(* CoDeSys 2.3.9.35 project: semaforo.pro *)
(* Author: Altus *)
(* Libraries: DU35x.lib 7.7.11 15:59:13, Navigation.lib 15.7.11 10:06:00, SysLibTargetVisu.lib 26.11.08 09:53:28, Standard.lib 26.11.08 09:46:20, Iecsfc.lib 26.11.08 09:46:14, SYSLIBCALLBACK.LIB 26.11.08 09:53:30 *)

(* PLC configuration (modules and I/O channels)
COM1 [COM1] node 0, in %IB0 out %QB0 {BaudRate = 115200; Paridade = Sem Paridade; StopBits = 1 Stop Bit; Modem = Sem RTS/CTS; Delay = 5}
  MODBUS Escravo [Escravo] node 0, in %IB0 out %QB0 {EnderecoModbus = 2}
COM2 [COM2] node 1, in %IB0 out %QB0 {BaudRate = 115200; Paridade = Sem Paridade; StopBits = 1 Stop Bit; Modem = Sem RTS/CTS; Delay = 5}
  Desabilitada [Desabilitado485] node 0, in %IB0 out %QB0
Barramento [Barramento] node 1, in %IB0 out %QB0
  Entradas [Entradas] node 0, in %IB0 out %QB0
    Entradas Digitais 0 [Entradas0] node 0, in %IW0 out %QB0
      I00 AT %IX0.0 [BitInput] I0.0
      I01 AT %IX0.1 [BitInput] I0.1
      I02 AT %IX0.2 [BitInput] I0.2
      I03 AT %IX0.3 [BitInput] I0.3
      I04 AT %IX0.4 [BitInput] I0.4
      I05 AT %IX0.5 [BitInput] I0.5
      I06 AT %IX0.6 [BitInput] I0.6
      I07 AT %IX0.7 [BitInput] I0.7
      I08 AT %IX0.8 [BitInput] I0.8
    Entradas Digitais 1 [Entradas1] node 0, in %IW1 out %QB0
      I10 AT %IX1.0 [BitInput] I1.0
      I11 AT %IX1.1 [BitInput] I1.1
      I12 AT %IX1.2 [BitInput] I1.2
      I13 AT %IX1.3 [BitInput] I1.3
      I14 AT %IX1.4 [BitInput] I1.4
      I15 AT %IX1.5 [BitInput] I1.5
      I16 AT %IX1.6 [BitInput] I1.6
      I17 AT %IX1.7 [BitInput] I1.7
      I18 AT %IX1.8 [BitInput] I1.8
    Entradas Digitais 2 [Entradas2] node 0, in %IW2 out %QB0
      I20 AT %IX2.0 [BitInput] I2.0
      I21 AT %IX2.1 [BitInput] I2.1
    Entradas Analógicas [EntradaAnalogica] node 0, in %IW4 out %QB0
      AI0 AT %IW4 [WordInput] AI0 {TipoAnalogica = Channel Disable; FiltroAnalogica = Filter 0 - AI=2ms  / AV=90ms; FundoEscala = 0}
      AI1 AT %IW5 [WordInput] AI1 {TipoAnalogica = Channel Disable; FiltroAnalogica = Filter 0 - AI=2ms  / AV=90ms; FundoEscala = 0}
      AI2 AT %IW6 [WordInput] AI2 {TipoAnalogica = Channel Disable; FiltroAnalogica = Filter 0 - AI=2ms  / AV=90ms; FundoEscala = 0}
      AI3 AT %IW7 [WordInput] AI3 {TipoAnalogica = Channel Disable; FiltroAnalogica = Filter 0 - AI=2ms  / AV=90ms; FundoEscala = 0}
    Entradas Rápidas [EntradasRapidas] node 1, in %IB16 out %QB0
      Bloco 0 [Bloco0] node 0, in %IB16 out %QB0
        Desabilitado [DesabilitadoBloco0] node 0, in %IB16 out %QB0
      Bloco 1 [Bloco1] node 1, in %IB16 out %QB0
        Desabilitado [DesabilitadoBloco1] node 0, in %IB16 out %QB0
      Entrada Configuravél Bloco 0 [EntradaConfiBloco0] node 2, in %IB16 out %QB0
        Contador 0 [EntradaConfContador0] node 0, in %IB16 out %QB0 {EntradaConfiguravelContador = Disable}
      Entrada Configuravél Bloco 1 [EntradaConfiBloco1] node 3, in %IB16 out %QB0
        Contador 2 [EntradaConfContador2] node 0, in %IB16 out %QB0 {EntradaConfiguravelContador = Disable}
  Saídas [Saidas] node 1, in %IB13 out %QB0
    Saídas Digitais 0 [Saidas0] node 0, in %IW0 out %QW0
      Q00 AT %QX0.0 [BitOutput] Q0.0
      Q01 AT %QX0.1 [BitOutput] Q0.1
      Q02 AT %QX0.2 [BitOutput] Q0.2
      Q03 AT %QX0.3 [BitOutput] Q0.3
      Q04 AT %QX0.4 [BitOutput] Q0.4
      Q05 AT %QX0.5 [BitOutput] Q0.5
      Q06 AT %QX0.6 [BitOutput] Q0.6
      Q07 AT %QX0.7 [BitOutput] Q0.7
    Saídas Digitais 1 [Saidas1] node 0, in %IW0 out %QW1
      Q10 AT %QX1.0 [BitOutput] Q1.0
      Q11 AT %QX1.1 [BitOutput] Q1.1
      Q12 AT %QX1.2 [BitOutput] Q1.2
      Q13 AT %QX1.3 [BitOutput] Q1.3
      Q14 AT %QX1.4 [BitOutput] Q1.4
      Q15 AT %QX1.5 [BitOutput] Q1.5
      Q16 AT %QX1.6 [BitOutput] Q1.6
      Q17 AT %QX1.7 [BitOutput] Q1.7
    Saídas Analógicas [SaidaAnalogica] node 0, in %IW0 out %QW3
      AO0 AT %QW3 [WordOutput] AO0 {TipoAnalogica = Channel Disable; FundoEscala = 0}
      AO1 AT %QW4 [WordOutput] AO1 {TipoAnalogica = Channel Disable; FundoEscala = 0}
    Saídas Rápidas [SaidasRapidas] node 1, in %IB0 out %QB10
      Saída Rápida 0 Desabilitada [DesabilitadoF0] node 0, in %IB0 out %QB10
      Saída Rápida 1 Desabilitada [DesabilitadoF1] node 1, in %IB0 out %QB10
    Saídas Comum de Contador [SaidasContador] node 2, in %IB0 out %QB10
      Saída do Bloco 0 Desabilitada [DesabilitadoSaidaBloco0] node 0, in %IB0 out %QB10
      Saída do Bloco 1 Desabilitada [DesabilitadoSaidaBloco1] node 1, in %IB0 out %QB10
Eventos Externos [Eventos] node 2, in %IB13 out %QB6
  Evento Temporizado [TimerEvent] node 0, in %IB13 out %QB6 {Intervalo = 10}
*)

(* Task configuration *)
TASK PRINCIPAL (PRIORITY := 1, INTERVAL := T#100ms);
	PLC_PRG();
END_TASK
TASK NAVIGATION (PRIORITY := 1, INTERVAL := T#20ms);
	NAVEGA();
END_TASK
TASK VISUALIZATION (PRIORITY := 1, INTERVAL := T#500ms);
	MAINTARGETVISU_PAINT_CODE
END_TASK
TASK KEYBOARD_USAGE (PRIORITY := 1, INTERVAL := T#20ms);
	MAINTARGETVISU_INPUT_CODE
END_TASK

(* POU PLC_PRG, LD *)
PROGRAM PLC_PRG
VAR
	t1: TON;
	t2: TON;
	t3: TON;
	t4: TON;
	t5: TON;
	t6: TON;
	v1: TON;
	a1: TON;
	ton1: TON;
	aux1: BOOL;
	taux: TON;
	vermelho_in AT %MW3: WORD;
	verde_in AT %MW4: WORD;
	amarelo_in : REAL := 4000;
	vermelho_out: TIME;
	verde_out: TIME;
	amarelo_out: TIME;
	RED: DWORD;
	Defeito: BOOL;
	td: TON;
	S_def: BOOL;
	td2: TON;
	S_def2: BOOL;
	t7: TON;
	t8: TON;
	t9: TON;
	t10: TON;
	t11: TON;
	t12: TON;
	td3: TON;
	td4: TON;
	auxv2: BOOL;
	a2: TON;
	auxa2: BOOL;
	aux_t7: BOOL;
	aux_t8: BOOL;
	aux_t9: BOOL;
	aux_t10: BOOL;
	t_aux11: BOOL;
	aux_t12: BOOL;
	bob: BOOL;
	sai: BOOL;
	tf: TON;
	tf2: TON;
	tf3: TON;
	vermelhor_in_2: REAL;
	verde_in_2: REAL;
	amarelo_in_2: REAL :=4000;
	vermelho_out_2: TIME;
	verde_out_2: TIME;
	amarelo_out_2: TIME;
	DEFEITO_SUP AT %MW7: WORD;
	DEFEITO_AUX:BOOL;
	LIGAR: BOOL;
	LIGAR_SUP AT %MW9: WORD;
END_VAR
VAR_INPUT
	SW1 AT %IX0.0: BOOL;
	SW2 AT %IX0.1: BOOL;
END_VAR
VAR_OUTPUT
	L1 AT %QX1.0: BOOL;
	L2 AT %QX1.1: BOOL;
	L3 AT %QX1.2: BOOL;
	L4 AT %QX1.3: BOOL;
	L5 AT %QX1.4: BOOL;
	L6 AT %QX1.5: BOOL;
	VERDE AT %QX1.6: BOOL;
	AMARELO AT %QX1.7: BOOL;
	aux: BOOL;
	M1 : BOOL;
	VERDE2: BOOL;
	AMARELO2: BOOL;
	M1_SUP AT %MW0: WORD;
	VERDE2_SUP AT %MW2: WORD;
	AMARELO2_SUP AT %MW1: WORD;
END_VAR
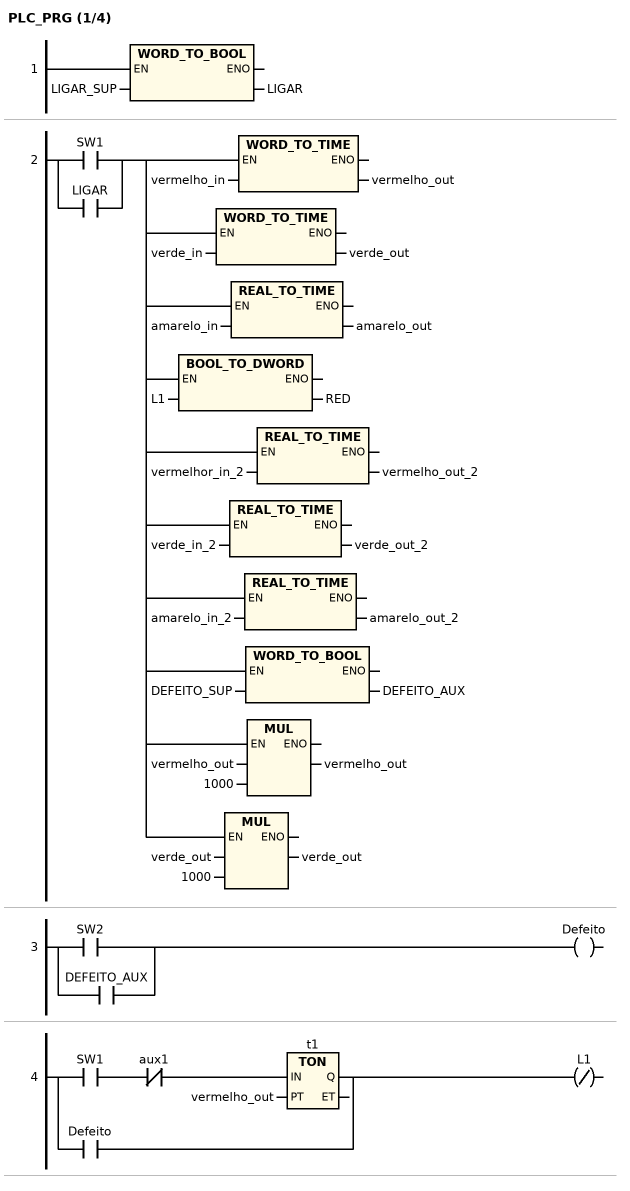
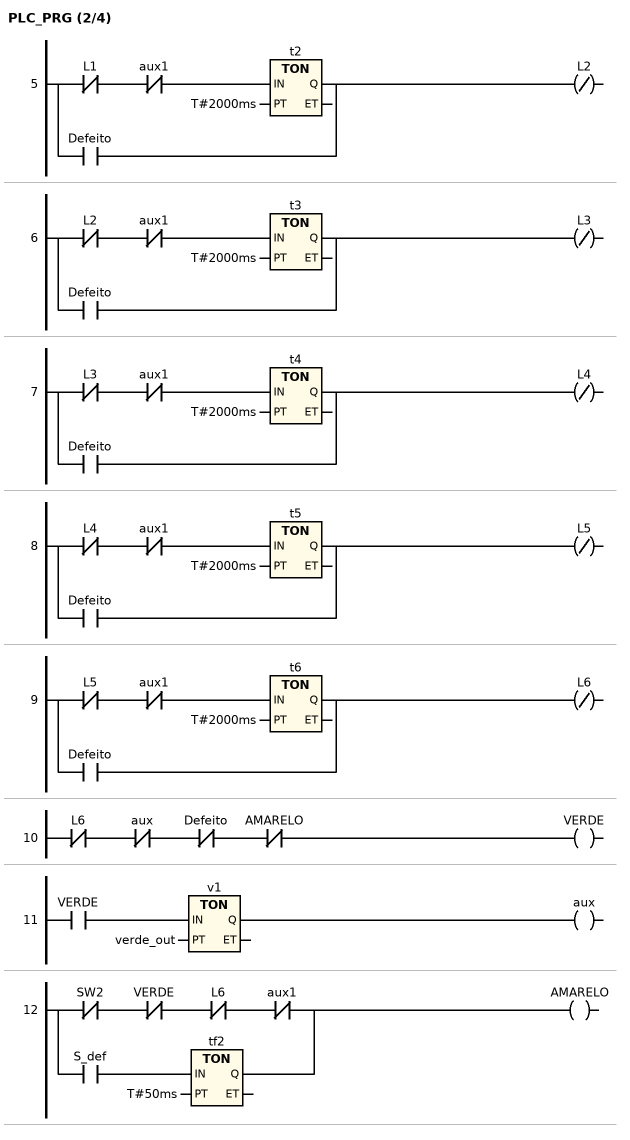
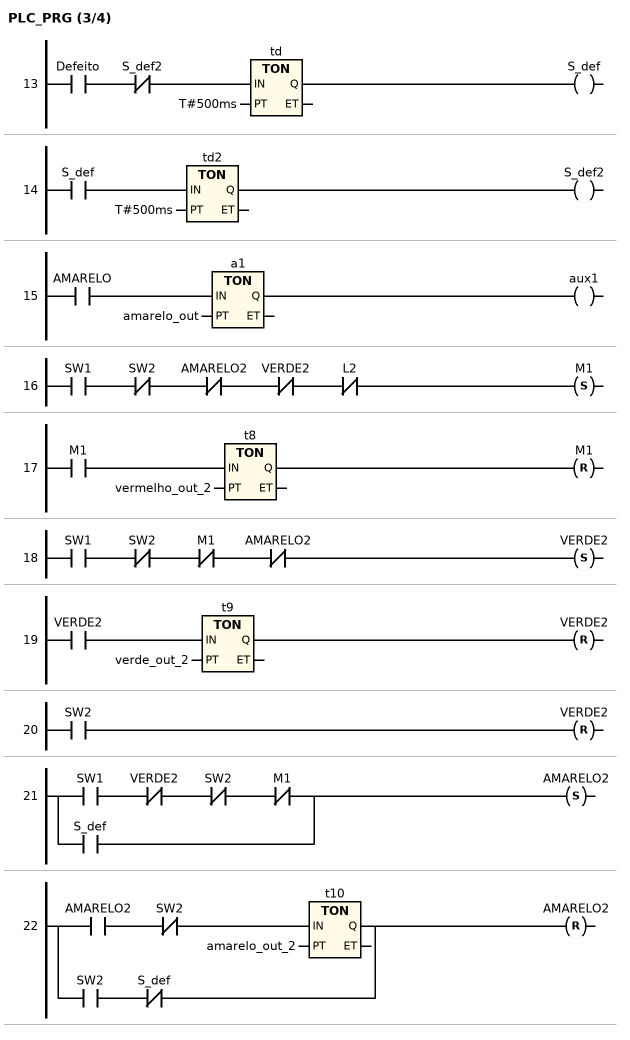
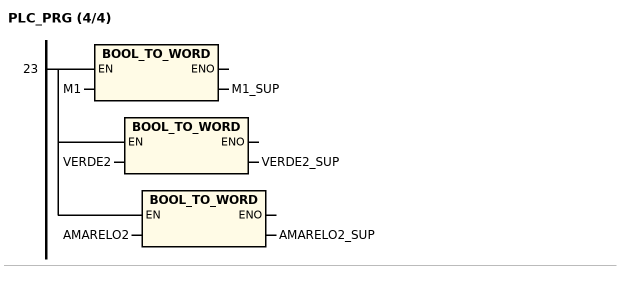
_LD_ (* Ladder Diagram *)
NETWORK 1
	*
		EN --- WORD_TO_BOOL(LIGAR_SUP) => LIGAR
NETWORK 2
	{ [SW1] | [LIGAR] }
		EN --- WORD_TO_TIME(vermelho_in) => vermelho_out
		EN --- WORD_TO_TIME(verde_in) => verde_out
		EN --- REAL_TO_TIME(amarelo_in) => amarelo_out
		EN --- BOOL_TO_DWORD(L1) => RED
		EN --- REAL_TO_TIME(vermelhor_in_2) => vermelho_out_2
		EN --- REAL_TO_TIME(verde_in_2) => verde_out_2
		EN --- REAL_TO_TIME(amarelo_in_2) => amarelo_out_2
		EN --- WORD_TO_BOOL(DEFEITO_SUP) => DEFEITO_AUX
		EN --- MUL(vermelho_out, 1000) => vermelho_out
		EN --- MUL(verde_out, 1000) => verde_out
NETWORK 3
	{ [SW2] | [DEFEITO_AUX] } --- (Defeito)
NETWORK 4
	{ [SW1] - [/aux1] - t1:TON(IN: *, PT: vermelho_out) | [Defeito] } --- (/L1)
NETWORK 5
	{ [/L1] - [/aux1] - t2:TON(IN: *, PT: T#2000ms) | [Defeito] } --- (/L2)
NETWORK 6
	{ [/L2] - [/aux1] - t3:TON(IN: *, PT: T#2000ms) | [Defeito] } --- (/L3)
NETWORK 7
	{ [/L3] - [/aux1] - t4:TON(IN: *, PT: T#2000ms) | [Defeito] } --- (/L4)
NETWORK 8
	{ [/L4] - [/aux1] - t5:TON(IN: *, PT: T#2000ms) | [Defeito] } --- (/L5)
NETWORK 9
	{ [/L5] - [/aux1] - t6:TON(IN: *, PT: T#2000ms) | [Defeito] } --- (/L6)
NETWORK 10
	[/L6] - [/aux] - [/Defeito] - [/AMARELO] --- (VERDE)
NETWORK 11
	[VERDE] - v1:TON(IN: *, PT: verde_out) --- (aux)
NETWORK 12
	{ [/SW2] - [/VERDE] - [/L6] - [/aux1] | [S_def] - tf2:TON(IN: *, PT: T#50ms) } --- (AMARELO)
NETWORK 13
	[Defeito] - [/S_def2] - td:TON(IN: *, PT: T#500ms) --- (S_def)
NETWORK 14
	[S_def] - td2:TON(IN: *, PT: T#500ms) --- (S_def2)
NETWORK 15
	[AMARELO] - a1:TON(IN: *, PT: amarelo_out) --- (aux1)
NETWORK 16
	[SW1] - [/SW2] - [/AMARELO2] - [/VERDE2] - [/L2] --- (S M1)
NETWORK 17
	[M1] - t8:TON(IN: *, PT: vermelho_out_2) --- (R M1)
NETWORK 18
	[SW1] - [/SW2] - [/M1] - [/AMARELO2] --- (S VERDE2)
NETWORK 19
	[VERDE2] - t9:TON(IN: *, PT: verde_out_2) --- (R VERDE2)
NETWORK 20
	[SW2] --- (R VERDE2)
NETWORK 21
	{ [SW1] - [/VERDE2] - [/SW2] - [/M1] | [S_def] } --- (S AMARELO2)
NETWORK 22
	{ [AMARELO2] - [/SW2] - t10:TON(IN: *, PT: amarelo_out_2) | [SW2] - [/S_def] } --- (R AMARELO2)
NETWORK 23
	*
		EN --- BOOL_TO_WORD(M1) => M1_SUP
		EN --- BOOL_TO_WORD(VERDE2) => VERDE2_SUP
		EN --- BOOL_TO_WORD(AMARELO2) => AMARELO2_SUP
_END_LD_
(* the same logic as Structured Text *)
(* Network 1 *)
LIGAR := WORD_TO_BOOL(LIGAR_SUP);
(* Network 2 *)
IF SW1 OR LIGAR THEN
	vermelho_out := WORD_TO_TIME(vermelho_in);
	verde_out := WORD_TO_TIME(verde_in);
	amarelo_out := REAL_TO_TIME(amarelo_in);
	RED := BOOL_TO_DWORD(L1);
	vermelho_out_2 := REAL_TO_TIME(vermelhor_in_2);
	verde_out_2 := REAL_TO_TIME(verde_in_2);
	amarelo_out_2 := REAL_TO_TIME(amarelo_in_2);
	DEFEITO_AUX := WORD_TO_BOOL(DEFEITO_SUP);
	vermelho_out := vermelho_out * 1000;
	verde_out := verde_out * 1000;
END_IF;
(* Network 3 *)
Defeito := SW2 OR DEFEITO_AUX;
(* Network 4 *)
t1(IN := SW1 AND NOT aux1, PT := vermelho_out);
L1 := NOT (t1.Q OR Defeito);
(* Network 5 *)
t2(IN := NOT L1 AND NOT aux1, PT := T#2000ms);
L2 := NOT (t2.Q OR Defeito);
(* Network 6 *)
t3(IN := NOT L2 AND NOT aux1, PT := T#2000ms);
L3 := NOT (t3.Q OR Defeito);
(* Network 7 *)
t4(IN := NOT L3 AND NOT aux1, PT := T#2000ms);
L4 := NOT (t4.Q OR Defeito);
(* Network 8 *)
t5(IN := NOT L4 AND NOT aux1, PT := T#2000ms);
L5 := NOT (t5.Q OR Defeito);
(* Network 9 *)
t6(IN := NOT L5 AND NOT aux1, PT := T#2000ms);
L6 := NOT (t6.Q OR Defeito);
(* Network 10 *)
VERDE := NOT L6 AND NOT aux AND NOT Defeito AND NOT AMARELO;
(* Network 11 *)
v1(IN := VERDE, PT := verde_out);
aux := v1.Q;
(* Network 12 *)
tf2(IN := S_def, PT := T#50ms);
AMARELO := NOT SW2 AND NOT VERDE AND NOT L6 AND NOT aux1 OR tf2.Q;
(* Network 13 *)
td(IN := Defeito AND NOT S_def2, PT := T#500ms);
S_def := td.Q;
(* Network 14 *)
td2(IN := S_def, PT := T#500ms);
S_def2 := td2.Q;
(* Network 15 *)
a1(IN := AMARELO, PT := amarelo_out);
aux1 := a1.Q;
(* Network 16 *)
IF SW1 AND NOT SW2 AND NOT AMARELO2 AND NOT VERDE2 AND NOT L2 THEN M1 := TRUE; END_IF;
(* Network 17 *)
t8(IN := M1, PT := vermelho_out_2);
IF t8.Q THEN M1 := FALSE; END_IF;
(* Network 18 *)
IF SW1 AND NOT SW2 AND NOT M1 AND NOT AMARELO2 THEN VERDE2 := TRUE; END_IF;
(* Network 19 *)
t9(IN := VERDE2, PT := verde_out_2);
IF t9.Q THEN VERDE2 := FALSE; END_IF;
(* Network 20 *)
IF SW2 THEN VERDE2 := FALSE; END_IF;
(* Network 21 *)
IF SW1 AND NOT VERDE2 AND NOT SW2 AND NOT M1 OR S_def THEN AMARELO2 := TRUE; END_IF;
(* Network 22 *)
t10(IN := AMARELO2 AND NOT SW2, PT := amarelo_out_2);
IF t10.Q OR SW2 AND NOT S_def THEN AMARELO2 := FALSE; END_IF;
(* Network 23 *)
M1_SUP := BOOL_TO_WORD(M1);
VERDE2_SUP := BOOL_TO_WORD(VERDE2);
AMARELO2_SUP := BOOL_TO_WORD(AMARELO2);
END_PROGRAM

(* POU NAVEGA, ST *)
PROGRAM NAVEGA
VAR
	ControleTelas : NAVIGATION;
	ListaTelas 	: ARRAY [0..30] OF STRING(10);
END_VAR
(* Adiciona a tela MAIN como tela principal *)
ListaTelas[0] := 'MAIN';

(* Ativa o controle automático de navegação somente pelo teclado *)
ControleTelas(ENABLE_UPDW := FALSE, VISU_LIST := ListaTelas, UP := FALSE , DOWN := FALSE);
END_PROGRAM
